FUNCTION_BLOCK INI (* Load and Store Data from settings.ini by Section and Key. Keys also present in the read-only settingsReadOnly.ini overlay cannot be modified via SET. *)
  (* Standard: 61499-2; Description: Copyright (c) 2024 HR Agrartechnik GmbH This program and the accompanying materials are made available under the terms of the Eclipse Public License 2.0 which is available at https://www.eclipse.org/legal/epl-2.0/ SPDX-License-Identifier: EPL-2.0 *)
  (* Version 3.2, 2026-08-01, Franz Höpfinger, HR Agrartechnik GmbH, read-only keys rejected by SET set STATUS to ERR_READ_ONLY, SETO is emitted when STATUS == OK, and SETOE otherwise *)
  (* Version 3.1, 2026-06-12, Franz Höpfinger, HR Agrartechnik GmbH, added Error Handling *)
  (* Version 3.0, 2025-04-14, Patrick Aigner, changed package *)
  (* Version 1.0, 2024-09-17, Franz Höpfinger, HR Agrartechnik GmbH *)
  PACKAGE eclipse4diac::storage;
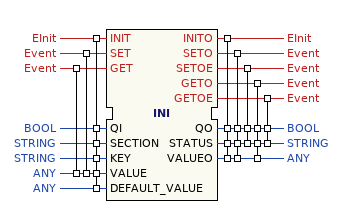
  EVENT_INPUT
    INIT : EInit WITH QI, SECTION, KEY, VALUE, DEFAULT_VALUE; (* Service Initialization *)
    SET WITH VALUE; (* set value for given key *)
    GET WITH VALUE; (* get value for given key *)
  END_EVENT
  EVENT_OUTPUT
    INITO : EInit WITH QO, STATUS, VALUEO; (* Initialization Confirm *)
    SETO WITH QO, STATUS, VALUEO; (* Confirmation of SET *)
    SETOE WITH QO, STATUS; (* Confirmation of SET in Error Case (see STATUS) *)
    GETO WITH QO, STATUS, VALUEO; (* Confirmation of GET *)
    GETOE WITH QO, STATUS; (* Confirmation of GET in Error Case (see STATUS) *)
  END_EVENT
  VAR_INPUT
    QI : BOOL; (* Event Input Qualifier *)
    SECTION : STRING; (* Section name. *)
    KEY : STRING; (* Key name. *)
    VALUE : ANY; (* The value to set. *)
    DEFAULT_VALUE : ANY; (* The value to read if there is noting in the settings.ini *)
  END_VAR
  VAR_OUTPUT
    QO : BOOL; (* Event Output Qualifier *)
    STATUS : STRING; (* Service Status *)
    VALUEO : ANY; (* The output value *)
  END_VAR
END_FUNCTION_BLOCK
